SUBAPPLICATION SubscribeEventHTTPFull (* Publish event using HTTP.  The consumer is encapsulated *)
  (* Standard: 61499-2; Description: Copyright (c) 2019 fortiss GmbH This program and the accompanying materials are made SPDX-License-Identifier: EPL-2.0 *)
  (* Version 1.0, 2019-11-12, Jose Cabral, fortiss GmbH *)
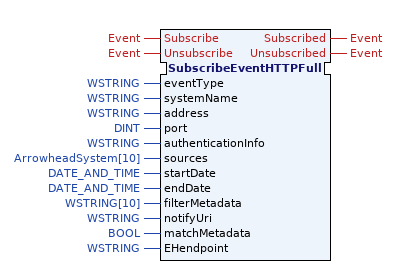
  EVENT_INPUT
    Subscribe;
    Unsubscribe;
  END_EVENT
  EVENT_OUTPUT
    Subscribed;
    Unsubscribed;
  END_EVENT
  VAR_INPUT
    eventType : WSTRING; (* Event type, similar to topics in MQTT *)
    systemName : WSTRING; (* Identification of the system *)
    address : WSTRING; (* Address of the offered services *)
    port : DINT; (* Port of the of the offered services *)
    authenticationInfo : WSTRING; (* Authentication info of the system *)
    sources : ARRAY [0..9] OF ArrowheadSystem; (* List of ArrowheadSystem the Subscriber wants to receive events from *)
    startDate : DATE_AND_TIME; (* If set, the Subscriber wants to receive events with timestamps after this date-time *)
    endDate : DATE_AND_TIME; (* If set, the Subscriber wants to receive events with timestamps before this date-time *)
    filterMetadata : ARRAY [0..9] OF WSTRING; (* Metadata about the events, which can be used for further filtering in format key=value *)
    notifyUri : WSTRING; (* The URL subpath where the Event Handler should sent the new events to *)
    matchMetadata : BOOL; (* Should the Event Handler filter events based on the metadata *)
    EHendpoint : WSTRING; (* Endpoint (IP:PORT/URI) of the Service Registry (not officially in the documentation, but it simplifies the FBs) *)
  END_VAR
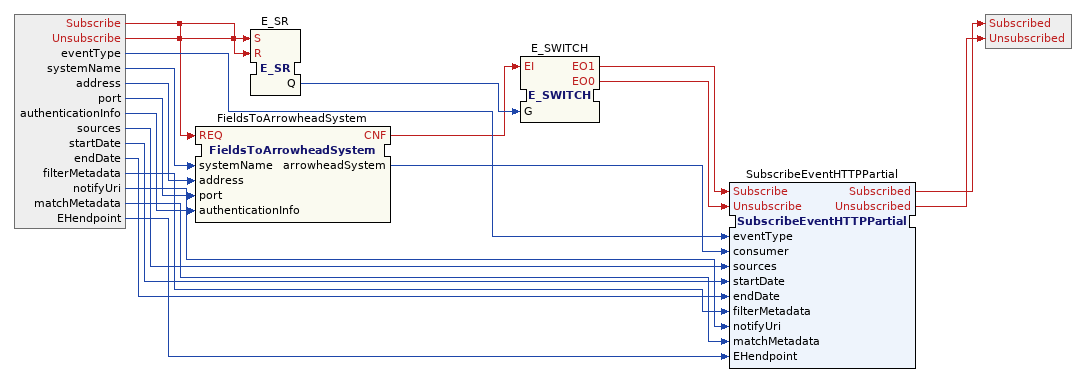
  FBS
    E_SWITCH : E_SWITCH;
    E_SR : E_SR;
    FieldsToArrowheadSystem : FieldsToArrowheadSystem;
  END_FBS
  SUBAPPS
    SubscribeEventHTTPPartial : SubscribeEventHTTPPartial;
  END_SUBAPPS
  EVENT_CONNECTIONS
    Subscribe TO E_SR.S;
    Unsubscribe TO E_SR.R;
    Unsubscribe TO FieldsToArrowheadSystem.REQ;
    Subscribe TO FieldsToArrowheadSystem.REQ;
    E_SWITCH.EO1 TO SubscribeEventHTTPPartial.Subscribe;
    E_SWITCH.EO0 TO SubscribeEventHTTPPartial.Unsubscribe;
    FieldsToArrowheadSystem.CNF TO E_SWITCH.EI;
    SubscribeEventHTTPPartial.Subscribed TO Subscribed;
    SubscribeEventHTTPPartial.Unsubscribed TO Unsubscribed;
  END_CONNECTIONS
  DATA_CONNECTIONS
    E_SR.Q TO E_SWITCH.G;
    systemName TO FieldsToArrowheadSystem.systemName;
    address TO FieldsToArrowheadSystem.address;
    port TO FieldsToArrowheadSystem.port;
    authenticationInfo TO FieldsToArrowheadSystem.authenticationInfo;
    eventType TO SubscribeEventHTTPPartial.eventType;
    FieldsToArrowheadSystem.arrowheadSystem TO SubscribeEventHTTPPartial.consumer;
    sources TO SubscribeEventHTTPPartial.sources;
    startDate TO SubscribeEventHTTPPartial.startDate;
    endDate TO SubscribeEventHTTPPartial.endDate;
    notifyUri TO SubscribeEventHTTPPartial.notifyUri;
    matchMetadata TO SubscribeEventHTTPPartial.matchMetadata;
    filterMetadata TO SubscribeEventHTTPPartial.filterMetadata;
    EHendpoint TO SubscribeEventHTTPPartial.EHendpoint;
  END_CONNECTIONS
END_SUBAPPLICATION
